TYPE Ffumatrixconfig :
STRUCT
	Enable : BOOL;
	FfuMatrix : ARRAY [0 .. Constants.speedMatrixSize] OF FfuSpeed;
END_STRUCT
END_TYPE

(* stored: Version 1.1.0.1, ProductVersion 3.1.4024.12
   DUT Ffumatrixconfig: Id {11ed2a13-50fd-4fd0-bb46-20d62a98ea5e} *)
